// TIA Portal V19 export
FUNCTION "TEST_O_ENDING_Fun" : Void   // FC204, LAD
// stored: SetENOAutomatically false
   VAR_TEMP   // added for the SCL form of the ladder/FBD networks
      _w1 : Bool;
   END_VAR
BEGIN

REGION Network 1
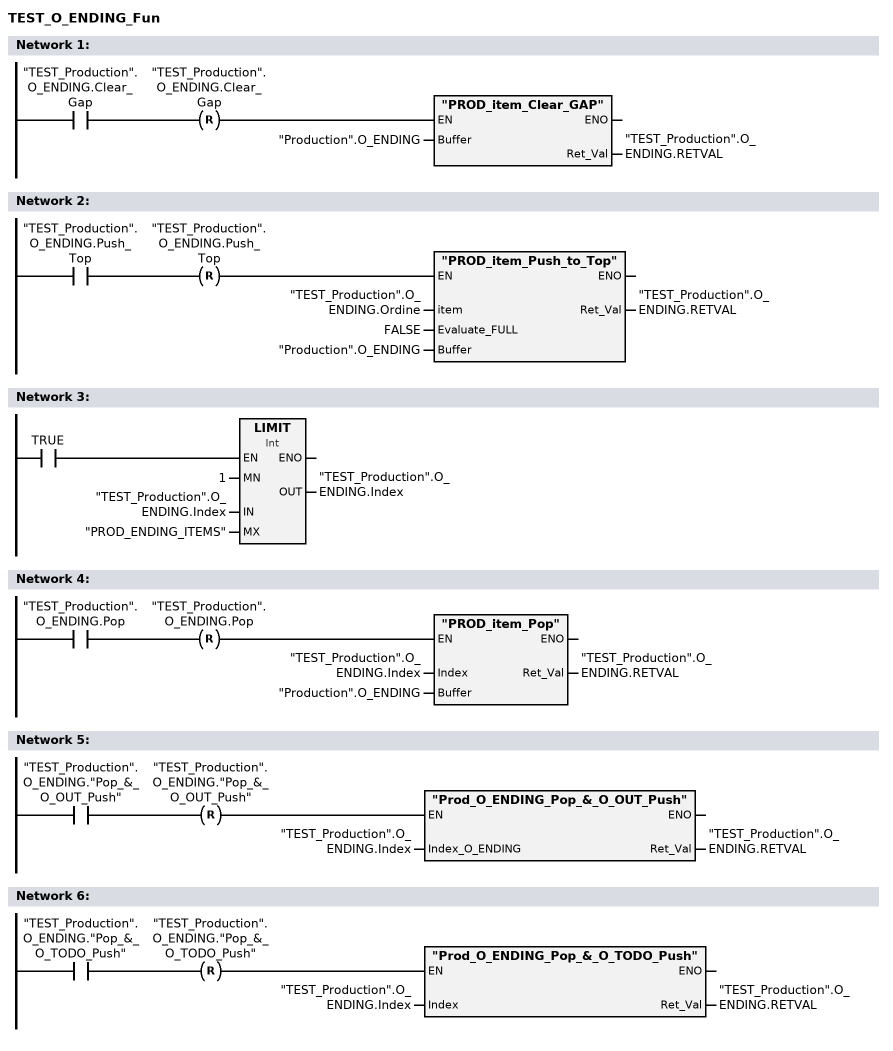
   RUNG wire#powerrail
      Contact( "TEST_Production".O_ENDING.Clear_Gap )
      R_Coil( "TEST_Production".O_ENDING.Clear_Gap )
      "PROD_item_Clear_GAP"(Buffer := "Production".O_ENDING, Ret_Val => "TEST_Production".O_ENDING.RETVAL)
   END_RUNG
   // the same network as SCL:
   #_w1 := "TEST_Production".O_ENDING.Clear_Gap;
   IF #_w1 THEN
       "TEST_Production".O_ENDING.Clear_Gap := FALSE;
       "TEST_Production".O_ENDING.RETVAL := "PROD_item_Clear_GAP"(Buffer := "Production".O_ENDING);
   END_IF;
END_REGION

REGION Network 2
   RUNG wire#powerrail
      Contact( "TEST_Production".O_ENDING.Push_Top )
      R_Coil( "TEST_Production".O_ENDING.Push_Top )
      "PROD_item_Push_to_Top"(item := "TEST_Production".O_ENDING.Ordine, Evaluate_FULL := FALSE, Buffer := "Production".O_ENDING, Ret_Val => "TEST_Production".O_ENDING.RETVAL)
   END_RUNG
   // the same network as SCL:
   #_w1 := "TEST_Production".O_ENDING.Push_Top;
   IF #_w1 THEN
       "TEST_Production".O_ENDING.Push_Top := FALSE;
       "TEST_Production".O_ENDING.RETVAL := "PROD_item_Push_to_Top"(item := "TEST_Production".O_ENDING.Ordine,
                               Evaluate_FULL := FALSE,
                               Buffer := "Production".O_ENDING);
   END_IF;
END_REGION

REGION Network 3
   RUNG wire#powerrail
      Contact( TRUE )
      { S7_Templates := "value_type := Int" } Limit(mn := 1, in := "TEST_Production".O_ENDING.Index, mx := "PROD_ENDING_ITEMS", out => "TEST_Production".O_ENDING.Index)
   END_RUNG
   // the same network as SCL:
   IF TRUE THEN
       "TEST_Production".O_ENDING.Index := LIMIT(MN := 1, IN := "TEST_Production".O_ENDING.Index, MX := "PROD_ENDING_ITEMS");
   END_IF;
END_REGION

REGION Network 4
   RUNG wire#powerrail
      Contact( "TEST_Production".O_ENDING.Pop )
      R_Coil( "TEST_Production".O_ENDING.Pop )
      "PROD_item_Pop"(Index := "TEST_Production".O_ENDING.Index, Buffer := "Production".O_ENDING, Ret_Val => "TEST_Production".O_ENDING.RETVAL)
   END_RUNG
   // the same network as SCL:
   #_w1 := "TEST_Production".O_ENDING.Pop;
   IF #_w1 THEN
       "TEST_Production".O_ENDING.Pop := FALSE;
       "TEST_Production".O_ENDING.RETVAL := "PROD_item_Pop"(Index := "TEST_Production".O_ENDING.Index,
                               Buffer := "Production".O_ENDING);
   END_IF;
END_REGION

REGION Network 5
   RUNG wire#powerrail
      Contact( "TEST_Production".O_ENDING."Pop_&_O_OUT_Push" )
      R_Coil( "TEST_Production".O_ENDING."Pop_&_O_OUT_Push" )
      "Prod_O_ENDING_Pop_&_O_OUT_Push"(Index_O_ENDING := "TEST_Production".O_ENDING.Index, Ret_Val => "TEST_Production".O_ENDING.RETVAL)
   END_RUNG
   // the same network as SCL:
   #_w1 := "TEST_Production".O_ENDING."Pop_&_O_OUT_Push";
   IF #_w1 THEN
       "TEST_Production".O_ENDING."Pop_&_O_OUT_Push" := FALSE;
       "TEST_Production".O_ENDING.RETVAL := "Prod_O_ENDING_Pop_&_O_OUT_Push"(Index_O_ENDING := "TEST_Production".O_ENDING.Index);
   END_IF;
END_REGION

REGION Network 6
   RUNG wire#powerrail
      Contact( "TEST_Production".O_ENDING."Pop_&_O_TODO_Push" )
      R_Coil( "TEST_Production".O_ENDING."Pop_&_O_TODO_Push" )
      "Prod_O_ENDING_Pop_&_O_TODO_Push"(Index := "TEST_Production".O_ENDING.Index, Ret_Val => "TEST_Production".O_ENDING.RETVAL)
   END_RUNG
   // the same network as SCL:
   #_w1 := "TEST_Production".O_ENDING."Pop_&_O_TODO_Push";
   IF #_w1 THEN
       "TEST_Production".O_ENDING."Pop_&_O_TODO_Push" := FALSE;
       "TEST_Production".O_ENDING.RETVAL := "Prod_O_ENDING_Pop_&_O_TODO_Push"(Index := "TEST_Production".O_ENDING.Index);
   END_IF;
END_REGION
END_FUNCTION
